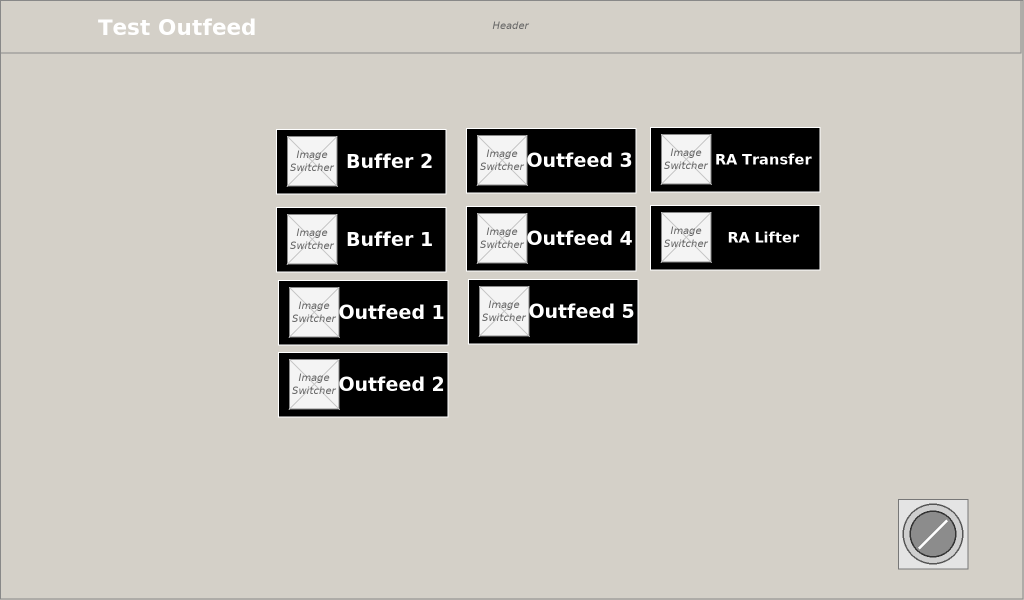
VISUALIZATION Test_Outfeed  // 1024x600
    Frame (0,-2 1021x55)
        shows Header()
    Label (95,15 250x25), "Test Outfeed"
    RotarySwitch (898,499 70x70), variable: HMI_GVL.bTestModeEnableOutfeed, behaviour: TOGGLE, style: Switch-RotarySwitch-Gray
    Group (276,129 182x65)
        toggle HMI_GVL.Test_PalletBuffer2_Fwd
        RoundedRectangle (0,0 170x65)
        Label (45,20 137x25), "Buffer 2"
        ImageSwitcher (11,7 50x50), variable: HMI_GVL.Test_PalletBuffer2_Fwd, behaviour: TOGGLE
    RoundedRectangle (276,207 170x65)
        toggle HMI_GVL.Test_PalletBuffer1_Fwd
    Label (321,227 137x25), "Buffer 1"
    ImageSwitcher (287,214 50x50), variable: HMI_GVL.Test_PalletBuffer1_Fwd, behaviour: TOGGLE
    RoundedRectangle (278,280 170x65)
        toggle HMI_GVL.Test_PalletOutfeed1_Fwd
    Label (323,300 137x25), "Outfeed 1"
    ImageSwitcher (289,287 50x50), variable: HMI_GVL.Test_PalletOutfeed1_Fwd, behaviour: TOGGLE
    RoundedRectangle (278,352 170x65)
        toggle HMI_GVL.Test_PalletOutfeed2_Fwd
    Label (323,372 137x25), "Outfeed 2"
    ImageSwitcher (289,359 50x50), variable: HMI_GVL.Test_PalletOutfeed2_Fwd, behaviour: TOGGLE
    RoundedRectangle (466,128 170x65)
        toggle HMI_GVL.Test_PalletOutfeed3_Fwd
    Label (511,148 137x25), "Outfeed 3"
    ImageSwitcher (477,135 50x50), variable: HMI_GVL.Test_PalletOutfeed3_Fwd, behaviour: TOGGLE
    RoundedRectangle (466,206 170x65)
        toggle HMI_GVL.Test_PalletOutfeed4_Fwd
    Label (511,226 137x25), "Outfeed 4"
    ImageSwitcher (477,213 50x50), variable: HMI_GVL.Test_PalletOutfeed4_Fwd, behaviour: TOGGLE
    RoundedRectangle (468,279 170x65)
        toggle HMI_GVL.Test_PalletOutfeed5_Fwd
    Label (513,299 137x25), "Outfeed 5"
    ImageSwitcher (479,286 50x50), variable: HMI_GVL.Test_PalletOutfeed5_Fwd, behaviour: TOGGLE
    RoundedRectangle (650,127 170x65)
        toggle HMI_GVL.Test_PalletRATransfer
    Label (695,147 137x25), "RA Transfer"
    ImageSwitcher (661,134 50x50), variable: HMI_GVL.Test_PalletRATransfer, behaviour: TOGGLE
    RoundedRectangle (650,205 170x65)
        tap HMI_GVL.Test_PalletRALifter
    Label (695,225 137x25), "RA Lifter"
    ImageSwitcher (661,212 50x50), variable: HMI_GVL.Test_PalletRALifter, behaviour: TOGGLE
END_VISUALIZATION

(* stored: Version 1.1.0.1, ProductVersion 3.1.4024.12
   Visu Test_Outfeed: Id {23b03dd1-866d-494e-b57c-58fdb0e99859} *)
